Staubli VAL3: OnF3.pgx

program OnF3()
begin
  call Prd:start()
  bUserRefresh=true
end
